TYPE sdd :
    UNION
    i : INT;
    END_UNION
END_TYPE

(* stored: Version 1.1.0.1, ProductVersion 3.1.4024.16
   DUT sdd: Id {9fd823d0-bf77-4c21-9de1-d351d266d6b8} *)
